PROGRAM MAIN
VAR

END_VAR


WareHousingExample();

LabelingExample();

//CamGearExample();

END_PROGRAM

(* stored: Version 1.1.0.1, ProductVersion 3.1.4024.11
   POU MAIN: Id {ce97d388-e861-4591-bddd-7771707f573f}, SpecialFunc None *)
